Staubli VAL3: CartesianForce.dtx

public num fx
public num fy
public num fz
public num frx
public num fry
public num frz
